{attribute 'linkalways'}
{attribute 'hide_all_locals'}
FUNCTION_BLOCK ValueLrealRead EXTENDS ValueBase IMPLEMENTS ValueRead
VAR
	thisValue : LREAL;
END_VAR

METHOD FB_init : BOOL
VAR_INPUT
	bInitRetains : BOOL; // if TRUE, the retain variables are initialized (warm start / cold start)
	bInCopyCode : BOOL;  // if TRUE, the instance afterwards gets moved into the copy code (online change)
END_VAR
_ValueType := __SYSTEM.TYPE_CLASS.TYPE_LREAL;
END_METHOD

METHOD Get : BOOL
VAR_INPUT
	destination : ANY;
END_VAR
Get := ConvertAnyType(thisAnyType, destination);
END_METHOD

METHOD GetAsString : T_MaxString
VAR_INPUT
END_VAR
GetAsString := TO_STRING(thisValue);
END_METHOD

METHOD GetAsType : BOOL
VAR_INPUT
	destination : __SYSTEM.AnyType;
END_VAR
GetAsType := ConvertAnyType(thisAnyType, destination);
END_METHOD

{attribute 'call_after_global_init_slot' := '1'}
{attribute 'call_after_online_change_slot' := '1'}
METHOD PROTECTED GetThisAnyType
VAR_INPUT
END_VAR
thisAnyType := ToAnyType(thisValue);
END_METHOD

END_FUNCTION_BLOCK

(* stored: Version 1.1.0.1, ProductVersion 3.1.4024.15
   POU ValueLrealRead: Id {7bbb62ae-f35c-4d8f-a9b3-e1cd293b29cb}, SpecialFunc None
   Method FB_init: Id {ac81c42f-d8fc-4c2d-897f-b50af6267b14}
   Method Get: Id {c695d588-c4b2-45c8-956d-6f9b3ebb2218}
   Method GetAsString: Id {e488a0bb-8605-44e1-9885-c332d07c2b85}
   Method GetAsType: Id {d4bab38f-a159-479b-843b-316f681562c1}
   Method GetThisAnyType: Id {0517e9a3-4e7f-42b0-b9dc-be44943d65f1} *)
